PROGRAM prgMain
VAR
	ADS_1: FB_ADS_Read;
	str_ADS_real_AverageRoomTemp: STRING(40);
	real_AverageRoomTemp	: REAL;											//{#lynus.ag#()}
	ton_Read_Delay: Ton;
END_VAR

// ADS Read out every minute
ton_Read_Delay( In:=TRUE AND NOT ton_Read_Delay.Q, 
				PT:=T#1M);
		
	
// start ADS read out of PLC Object ZVG
IF ton_Read_Delay.Q THEN
	str_ADS_real_AverageRoomTemp:='prgMain.real_AverageRoomTemp';
	ADS_1(	udintWriteLength:=SIZEOF(str_ADS_real_AverageRoomTemp),
			udintReadLength:=SIZEOF(real_AverageRoomTemp),
			dwSourceAddr:=ADR(str_ADS_real_AverageRoomTemp),
			dwDestAddr:=ADR(real_AverageRoomTemp),
			strNETid:='5.109.229.195.1.1');		// AMS NetID Object ZVG
END_IF

real_AverageRoomTemp := INT_TO_REAL(REAL_TO_INT(real_AverageRoomTemp*1000))/1000;

END_PROGRAM

(* stored: Version 1.1.0.1, ProductVersion 3.1.4024.11
   POU prgMain: Id {09755b01-d80b-414a-9783-185acd4cb0f4}, SpecialFunc None *)
